INTERFACE ITF_BaseTopElement_HMI_Connector EXTENDS ITF_BaseTopElement_HMI_Connector_View, ITF_BaseTopElement_HMI_Connector_Command

END_INTERFACE

(* stored: Version 1.1.0.1
   Itf ITF_BaseTopElement_HMI_Connector: Id {b063fadc-5c9f-0348-3cd4-53e9e9f7e38c} *)
